TYPE strQueueContentDetail :
	STRUCT
		uiPrio			: UINT;				(* Option Sendepriorität *)
		uiMsgHandle 	: UDINT;			(* unique msg handle,  *)
		aDATA			: ARRAY [0..Sewts_TCP.MAX_QueueData] OF BYTE ;	(* Data *)
		uiDATA			: UDINT;			(* Length of data from pointer reference*)	
	END_STRUCT
END_TYPE

(* stored: Version 1.1.0.1, ProductVersion 3.1.4024.12
   DUT strQueueContentDetail: Id {aa7da90c-8820-432d-b6bd-a6be3e69fc6e} *)
